# EPICS substitutions: ecmcApp/Db/el7037.substitutions
file "el7037.template"
{
pattern
{P,     PORT,   SLAVE_POS, STM_STAT,   STM_CNTRL,   VEL_SET,           ENC_STAT,   ENC_POS,  LATCH_POS      }
{IOC2:, MC_CPU1 7,         STM_STATUS, STM_CONTROL, VELOCITY_SETPOINT, ENC_STATUS, POSITION, LATCH_POSITION }
{IOC2:, MC_CPU1 8,         STM_STATUS, STM_CONTROL, VELOCITY_SETPOINT, ENC_STATUS, POSITION, LATCH_POSITION }
}
